INTERFACE I_DigitalOutput EXTENDS I_Channel

PROPERTY P_Value : bool
SET
END_SET
END_PROPERTY

END_INTERFACE

(* stored: Version 1.1.0.1
   Itf I_DigitalOutput: Id {3250afe1-4ca3-08ac-0e0d-69e5fb319b06}
   Property P_Value: Id {2aa110a8-71af-0218-2b6c-57a543435824}
   Set Set: Id {181a6780-dbcc-06e1-3994-44e2ca8c955e} *)
